// SIMATIC S7-200 project (STEP 7-Micro/WIN), CPU 216 REL 01.02

SYMBOL_TABLE USR1
Always_On        SM0.0    // This bit is always on.
First_Scan_On    SM0.1    // This bit is on for the first scan cycle only.
HSC0_Ctrl        SMB37    // This byte enables you to control the operation of high-speed counter 0.
HSC0_CV          SMD38    // New current value of high-speed counter 0. SMB38 is the most significant byte.
HSC0_PV          SMD42    // New preset value of high-speed counter 0. SMB42 is the most significant byte.
PLS0_Ctrl        SMB67    // Controls pulse train output & pulse width modulation functions for output Q0.0.
PLS0_Cycle       SMW68    // Cycle time value, pulse train or pls. width modulation output 0. SMB68 is MSB.
PTO0_PC          SMD72    // Pulse count value of pulse train output 0. SMB72 is the most significant byte.
END_SYMBOL_TABLE

SYMBOL_TABLE 
USS_LOW_V        VD1000
USS_HIGH_V       VD1004
USS_TIME_OUT     VW1008
USS_I_LINE       VW1010
USS_DAT_PTR0     VD1012
USS_ACT_DRV0     VD1016
USS_CUR_DRV0     VD1020
USS_P0           V1024.0
USS_REQ_SNT0     V1024.1
USS_RETRY_P0     VB1025
USS_ERR_CODE     VB1026
USS_CS_D0        VD1027
USS_CS_W0        VW1027
USS_CS_W2        VW1029
USS_CS_B0        VB1027
USS_CS_B1        VB1028
USS_POLL_BUF     VB1031
USS_XMT_0        VB1046
USS_XMT_ADR0     VB1049
USS_X_STWD       VD1056
USS_X_BCC        VB1060
USS_X_DW1        VD1047
USS_X_DW5        VD1051
USS_X_DW9        VD1055
USS_X_DB13       VB1059
USS_RCV_BUF0     VB1061
USS_R_STX        VB1062
USS_R_LGE        VB1063
USS_R_ADR        VB1064
USS_R_STWD       VD1071
USS_R_DW1        VD1062
USS_R_DW5        VD1066
USS_R_DW9        VD1070
USS_R_W13        VW1074
USS_STAT_TAB     VB1076
USS_ADR_P0       VB1396
END_SYMBOL_TABLE

ORGANIZATION_BLOCK MAIN:OB1
TITLE= Tip004B
// 题目： 怎样使用高速计数器
// ***概述***
// 本例叙述SIMATIC S7-200的高速计数器（HSC）的一种组态功能。对来自传感
// 器（如编码器）信号的处理，高速计数器可采用多种不同的组态功能
// 本例用脉冲输出（PLS）来为HSC产生高速计数信号，PLS可以产生脉冲串和脉
// 宽调制信号，例如用来控制伺服电机。既然利用脉冲输出，必须选用
// CPU214/DC/DC/DC
// 下面这个例子，展示了用HSC和脉冲输出构成一个简单的反馈回路，怎样编制
// 一个程序来实现反馈功能
// 
// ***程序和注释***
// 本例描述了S7-200 DC/DC/DC的高速计数器（HSC)的功能。HSC计数速度比PLC扫
// 描时间快的多,采用集成在S7-212中的2kHz的软件计数器进行计数。S7-214除了
// 有2kHz的计数器外,还有两个7kHz的硬件计数器，总的来说，每个高速计数器需要
// 10个字节内存用来存控制位、当前值、设定值、状态位。
// 本程序长度为91个字
// 
BEGIN
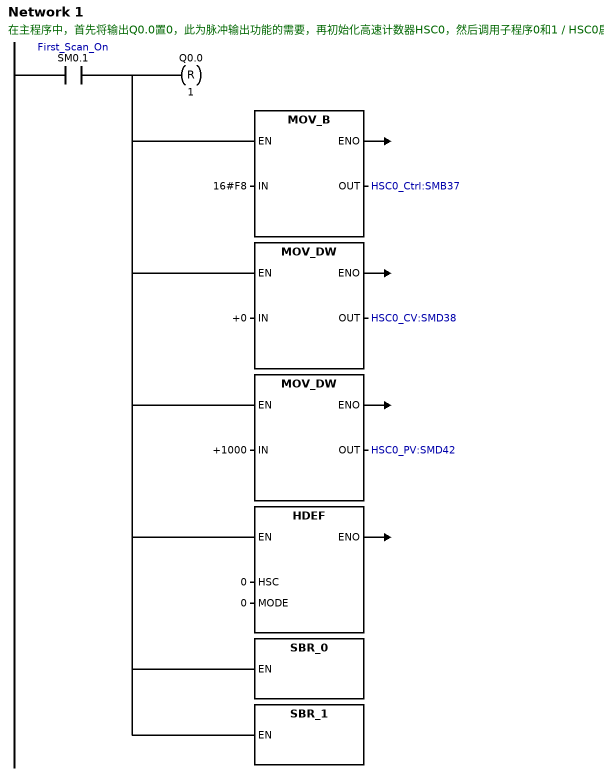
Network 1
// 在主程序中，首先将输出Q0.0置0，此为脉冲输出功能的需要，再初始化高速计数器HSC0，然后调用子程序0和1
// HSC0启动后具有下列特性：可更新CV和PV值，正向计数当脉冲输出数达到SMD72中规定的数后，程序就终止
// 首次扫描标志（SM0.1=1)
//脉冲串输出Q0.0复位（Q0.0=0).
// 装载HSC0的控制位
// HSC0当前值（CV)为0。
// HSCO的第一次设定值（PV)为1000
// HSC0定义模式0
// 调用子程序0。
// 调用子程序1。
LD     First_Scan_On:SM0.1
R      Q0.0, 1
MOVB   16#F8, HSC0_Ctrl:SMB37
MOVD   +0, HSC0_CV:SMD38
MOVD   +1000, HSC0_PV:SMD42
HDEF   0, 0
CALL   SBR_0:SBR0
CALL   SBR_1:SBR1
Network 2 //  主程序结束
//  MEND
// 
END_ORGANIZATION_BLOCK

SUBROUTINE_BLOCK SBR_0:SBR0
TITLE=
BEGIN
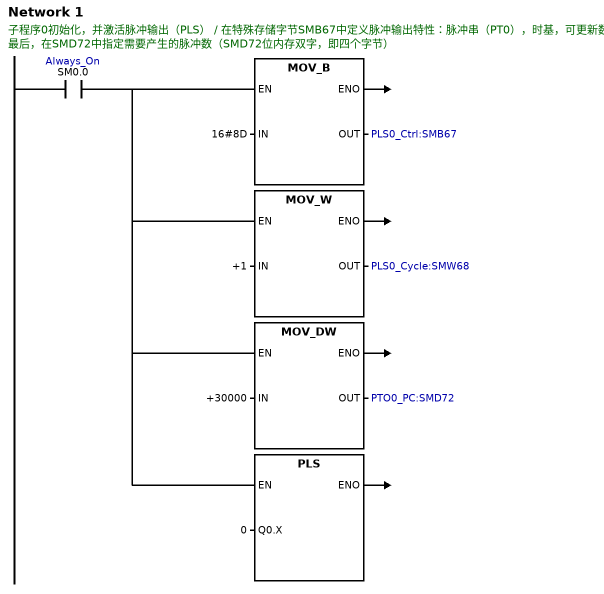
Network 1
// 子程序0初始化，并激活脉冲输出（PLS）
// 在特殊存储字节SMB67中定义脉冲输出特性：脉冲串（PT0），时基，可更新数值，激活PLS
// SMW68定义脉冲周期，其值为时基的倍数
// 最后，在SMD72中指定需要产生的脉冲数（SMD72位内存双字，即四个字节）
// 装载脉冲输出（PLS0)的控制位：PT0,时基
// 1ms，可更新，激活
// 脉冲周期1ms。
// 产生30000个脉冲。
// 起动脉冲输出（PLS0),从输出端Q0.0输出脉冲
LD     Always_On:SM0.0
MOVB   16#8D, PLS0_Ctrl:SMB67
MOVW   +1, PLS0_Cycle:SMW68
MOVD   +30000, PTO0_PC:SMD72
PLS    0
Network 2 // 子程序0结束
//  RET
// 
END_SUBROUTINE_BLOCK

SUBROUTINE_BLOCK SBR_1:SBR1
TITLE=
BEGIN
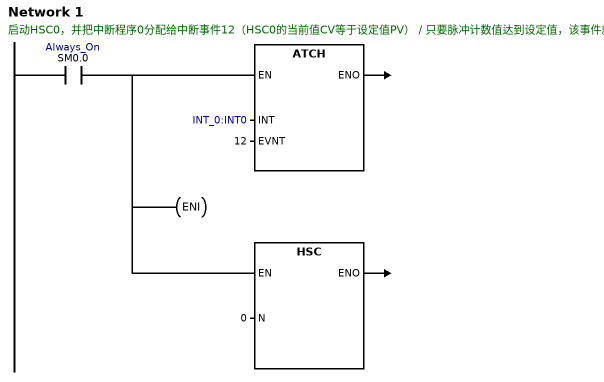
Network 1
// 启动HSC0，并把中断程序0分配给中断事件12（HSC0的当前值CV等于设定值PV）
// 只要脉冲计数值达到设定值，该事件就会发生
// 允许中断
//把中断程序0分配给中断事件12（HSC0的当前值CV等于设定值PV）
//允许中断 
// 按主程序中对HSC0的初始组态特性，起动HSC0。Start HSC0.
LD     Always_On:SM0.0
ATCH   INT_0:INT0, 12
ENI
HSC    0
Network 2 //  子程序1结束
//  RET
// 
END_SUBROUTINE_BLOCK

INTERRUPT_BLOCK INT_0:INT0
TITLE=
BEGIN
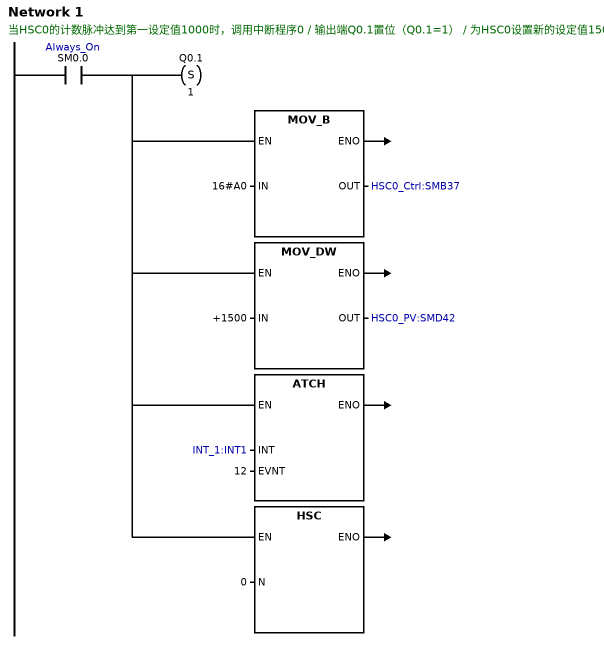
Network 1
// 当HSC0的计数脉冲达到第一设定值1000时，调用中断程序0
// 输出端Q0.1置位（Q0.1=1）
// 为HSC0设置新的设定值1500（第二设定值）
// 用中断程序1取代中断程序0，分配给中断事件12（HSC0的CV=PV）
// Load SM0.0.
// 输出端Q0.1置位（Q0.1=1） 
// 重置HSC0的控制位，仅更新设定值（PV）
// 为HSC0设置新的设定值1500（第二设定值）
// 用中断程序1取代中断程序0，分配给中断事件12  Attach interrupt event 12 to
// 起动HSC0,为其装载新的设定值 
LD     Always_On:SM0.0
S      Q0.1, 1
MOVB   16#A0, HSC0_Ctrl:SMB37
MOVD   +1500, HSC0_PV:SMD42
ATCH   INT_1:INT1, 12
HSC    0
Network 2 //  中断程序0结束
//  RETI
// 
END_INTERRUPT_BLOCK

INTERRUPT_BLOCK INT_1:INT1
TITLE=
BEGIN
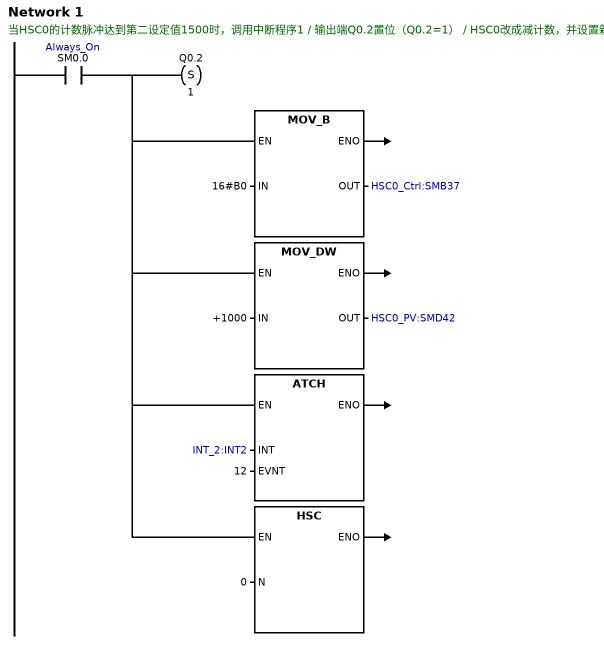
Network 1
// 当HSC0的计数脉冲达到第二设定值1500时，调用中断程序1
// 输出端Q0.2置位（Q0.2=1）
// HSC0改成减计数，并设置新的设定值1000（第三设定值）
// 用中断程序2取代中断程序1，分配给中断事件12（HSC0的CV=PV）
//输出端Q0.2置位（Q0.2=1） 
// 重置HSC0的控制位，更新设定值，并改成减计
//数（反向计数）
// HSC0的下一个设定值为1000（第三设定值）
// 用中断程序2取代中断程序1，分配给中断事件12 
// 起动HSC0,为其装载新的设定值和方向。
LD     Always_On:SM0.0
S      Q0.2, 1
MOVB   16#B0, HSC0_Ctrl:SMB37
MOVD   +1000, HSC0_PV:SMD42
ATCH   INT_2:INT2, 12
HSC    0
Network 2 //  中断程序1结束
//  RETI
// 
END_INTERRUPT_BLOCK

INTERRUPT_BLOCK INT_2:INT2
TITLE=
BEGIN
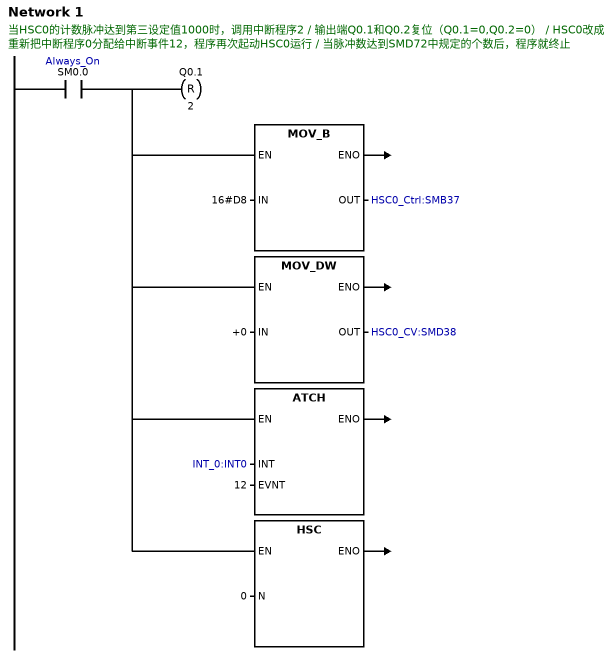
Network 1
// 当HSC0的计数脉冲达到第三设定值1000时，调用中断程序2
// 输出端Q0.1和Q0.2复位（Q0.1=0,Q0.2=0）
// HSC0改成加计数，并将当前计数值置为0，而设定值PV保持不变（1000）
// 重新把中断程序0分配给中断事件12，程序再次起动HSC0运行
// 当脉冲数达到SMD72中规定的个数后，程序就终止
// 输出端Q0.1和Q0.2复位（Q0.1=0,Q0.2=0） 
// 重置HSC0的控制位，更新CV，并改成正向计
// 数（增计数）
// HSC0的当前值复位（CV=0）
// 把中断程序0分配给中断事件12 
// 重新起动HSC 0. 
LD     Always_On:SM0.0
R      Q0.1, 2
MOVB   16#D8, HSC0_Ctrl:SMB37
MOVD   +0, HSC0_CV:SMD38
ATCH   INT_0:INT0, 12
HSC    0
Network 2 // 中断程序2结束
//  RETI				
// 
END_INTERRUPT_BLOCK
